PROGRAM MQTT
VAR
END_VAR

END_PROGRAM

(* stored: Version 1.1.0.1, ProductVersion 3.1.4024.12
   POU MQTT: Id {22a2f25d-52ae-4956-8afe-fe8eb2daff36}, SpecialFunc None *)
